TYPE ST_HMIEButton_HMI :
STRUCT
	bActive		: BOOL;
	bVisible	: BOOL;
	bEnable		: BOOL;
	bPushed		: BOOL;
END_STRUCT
END_TYPE

(* stored: Version 1.1.0.1
   DUT ST_HMIEButton_HMI: Id {dd614e4e-0bdc-0845-350f-74ce1aed1e8e} *)
